(* CoDeSys 2.3.9.37 project: Cap10_1_Res.pro *)
(* Libraries: STANDARD.LIB 4.10.05 12:14:46 *)

(* Global variable list: Globale_Variablen *)
VAR_GLOBAL

	(*Entradas*)
	Start : BOOL;
	ControlOK : BOOL;

      (*Salidas*)
	Warning : BOOL;
	Stop : BOOL;
END_VAR

(* POU PLC_PRG, FBD *)
PROGRAM PLC_PRG
VAR

	Trig1: R_TRIG;
	Trig2: F_TRIG;
	Timer1: TOF;
	Timer2: TON;

END_VAR
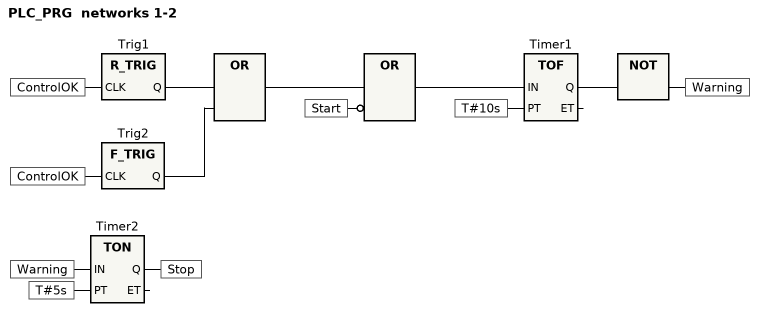
_FBD_ (* Function Block Diagram *)
NETWORK 1
	NOT Timer1:TOF(IN: OR(OR(Trig1:R_TRIG(CLK: ControlOK), Trig2:F_TRIG(CLK: ControlOK)), NOT Start), PT: T#10s) => Warning
NETWORK 2
	Timer2:TON(IN: Warning, PT: T#5s) => Stop
_END_FBD_
(* the same logic as Structured Text *)
(* Network 1 *)
Trig1(CLK := ControlOK);
Trig2(CLK := ControlOK);
Timer1(IN := (Trig1.Q OR Trig2.Q) OR NOT Start, PT := T#10s);
Warning := NOT Timer1.Q;
(* Network 2 *)
Timer2(IN := Warning, PT := T#5s);
Stop := Timer2.Q;
END_PROGRAM

(* Visualisation Observation
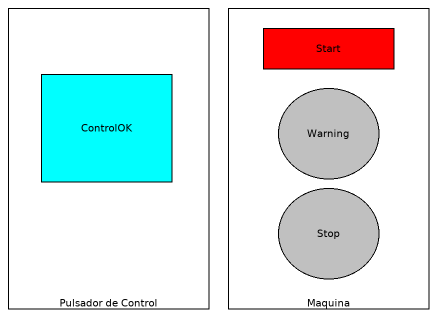
rectangle at (230,10)-(431,311): text "Maquina"
rectangle at (10,10)-(211,311): text "Pulsador de Control"
rectangle at (43,76)-(174,184): text "ControlOK"; alarm colour if ControlOK; toggles ControlOK
ellipse at (280,90)-(381,181): text "Warning"; alarm colour if Warning
ellipse at (280,190)-(381,281): text "Stop"; alarm colour if Stop
rectangle at (265,30)-(396,71): text "Start"; alarm colour if Start; toggles Start
*)
